Universal Robots PolyScope program: motiontest.urp

Program motiontest (installation=cube_dev1 directory=/programs createdIn=5.11.5.1010327 lastSavedIn=5.11.5.1010327 robotSerialNumber=20215500677)
Calibrated DH parameters: a=[0.000204, -0.239222, -0.391845, -0.000001, 0.000022, 0]; d=[0.162722, -355.808559, 353.37206, 2.570385, 0.099741, 0.099629]; alpha=[1.571124, 0.000988, 0.008295, 1.568963, -1.570303, 0]; deltaTheta=[0, -0.973091, 7.204745, 0.05153, 0, 0]
BeforeStart
  Script file /programs/cube/set_conveyor_params.script
    | def Set_Conveyor_Params(velocity, acceleration):
    | modbus_set_output_register("VELOCITY", velocity, False)
    | modbus_set_output_register("ACCELERATION", acceleration, False)
    | end
  Script file /programs/cube/set_motion_mode.script
    | def Set_Motion_Mode(modeString):
    |   if modeString == "distance":
    |     modbus_set_output_register("MOTION_MODE", 0, False)
    |   elif modeString == "position":
    |     modbus_set_output_register("MOTION_MODE", 1, False)
    |   elif modeString == "continuous":
    |     modbus_set_output_register("MOTION_MODE", 2, False)
    |   elif modeString == "idle":
    |     modbus_set_output_register("MOTION_MODE", 3, False)
    |   else:
    |     modbus_set_output_register("MOTION_MODE", 3, False)
    |   end
    | end
  Script file /programs/cube/position_move.script
    | def Move_Position(position):
    |   Set_Motion_Mode("position")
    |   modbus_set_output_register("POSITION", position, False)
    |   Set_Request_Id()
    |   sleep(.01)
    | end
  Script file /programs/cube/distance_move.script
    | def Move_Distance(distance):
    |   Set_Motion_Mode("distance")
    |   distance = Inches_To_Steps(distance)
    |   if distance < 0:
    |   distance = distance * -1
    |   modbus_set_output_signal("DIRECTION", False, False)
    |   else:
    |   modbus_set_output_signal("DIRECTION", True, False)
    |   end
    |   modbus_set_output_register("DISTANCE", distance, False)
    |   Set_Request_Id()
    |   sleep(.2)
    | end
  Script file /programs/cube/mm_move.script
    | def Conveyor_Move_mm(distance):
    |   Set_Motion_Mode("distance")
    |   distance = mm_to_steps(distance)
    |   if distance < 0:
    |   distance = distance * -1
    |   modbus_set_output_signal("DIRECTION", False, False)
    |   else:
    |   modbus_set_output_signal("DIRECTION", True, False)
    |   end
    |   modbus_set_output_register("DISTANCE", distance, False)
    |   Set_Request_Id()
    |   sleep(.05)
    | end
  Script file /programs/cube/continuous_move.script
    | def Move_Continuous(direction):
    |   Set_Motion_Mode("continuous")
    |   if direction == "forward":
    |   modbus_set_output_signal("DIRECTION", True, False)
    |   else:
    |   modbus_set_output_signal("DIRECTION", False, False)
    |   end
    |   Set_Request_Id()
    | end
  Script file /programs/cube/idle_move.script
    | def Move_Idle():
    |   Set_Motion_Mode("idle")
    |   Set_Request_Id()
    | end
  Script file /programs/cube/request_id.script
    | def Set_Request_Id():
    | id = floor(random()*65000)
    | modbus_set_output_register("REQUEST_ID", id, False)
    | end
  Script file /programs/cube/steps_per_inch.script
    | def Inches_To_Steps(distance):
    | mm = distance*25.4
    | return mm_to_steps(mm)
    | end
  Script file /programs/cube/mm_to_steps.script
    | def mm_to_steps(distance):
    | teeth = 28
    | pitch = 2
    | degreesPerStep = 1.8
    | microsteps = 8
    | adjustment = 400/381
    | microStepsPerMm = 360 / teeth  / degreesPerStep / pitch * microsteps * adjustment
    | return floor(distance * microStepsPerMm)
    | end
  Script: Set_Conveyor_Params(1600, 16000)
  Script: Move_Idle()
  Script file /programs/select_job.script
    | def read_job():
    | job = modbus_get_signal_status("JOB", False)
    | #1 - cube, 2 - browser,  3 - 45
    | #4 - stereocab 2, 5 - sc 3, 6 - sc4
    | if job == 1:
    |   width = 362
    |   height = 362
    |   depth = 349
    | elif job == 2:
    |   width = 362
    |   height = 362
    |   depth = 235
    | elif job == 3:
    |   width = 724
    |   height = 235
    |   depth = 349
    | elif job == 4:
    |   width = 724
    |   height = 235
    |   depth = 349
    | elif job == 5:
    |   width = 1086
    |   height = 235
    |   depth = 349
    | elif job == 1:
    |   width = 1148
    |   height = 235
    |   depth = 349
    | end
    | end
  loaded := 0
  MoveJ speed 60 deg/s, acceleration 80 deg/s^2 (useActiveTCP=false) tcp=SandTCP; feature=Base
    Waypoint Waypoint_1: TCP in base x=-330.988 y=207.997 z=636.996 mm, rx=0.0399 ry=-0.0211 rz=-2.2331 rad; joints [-56.152, -81.08, 119.99, 96.099, -76.463, -167.945] deg; TCP offset x=1.003 y=125.541 z=104.154 mm, rx=-0.7854 ry=0 rz=0 rad
Robot Program (runOnlyOnce=true)
  Script: read_job()
  Script: Conveyor_Move_mm(width)
  Wait Condition expression=SERVER_STATE == 1
  Script: Conveyor_Move_mm(-width)
  Wait Condition expression=SERVER_STATE == 1
